{attribute 'linkalways'} 
{attribute 'no_explicit_call' := 'This FB is a CLASS and must be accessed using methods or properties'}
{attribute 'enable_dynamic_creation'}
FUNCTION_BLOCK FINAL ABS_ULINT EXTENDS Node
VAR
	in : _ULINT(0);
	out : _ULINT(0);
END_VAR

METHOD PUBLIC Clone : I_Node
VAR
	pNode : POINTER TO ABS_ULINT;
END_VAR
pNode := __NEW(ABS_ULINT);
Clone := pNode^;
END_METHOD

METHOD FB_init : BOOL
VAR_INPUT
	bInitRetains : BOOL; // if TRUE, the retain variables are initialized (warm start / cold start)
	bInCopyCode : BOOL;  // if TRUE, the instance afterwards gets moved into the copy code (online change)
END_VAR
AddInput('in',THIS^.in);
AddOutput('out', THIS^.out);
END_METHOD

METHOD PROTECTED OnExecute
VAR
END_VAR
out.Value := ABS(in.Value);
END_METHOD

END_FUNCTION_BLOCK

(* stored: Version 1.1.0.1, ProductVersion 3.1.4024.15
   POU ABS_ULINT: Id {d9e94608-85d9-4704-aef5-600e84c92692}, SpecialFunc None
   Folder Constructor: Id {b89a9a35-a5c0-4751-a23a-8c3e69466e39}
   Method Clone: Id {8666aac5-0a1a-49e8-aae3-2f59925bd958}
   Method FB_init: Id {30dfa24d-4c2c-43c3-8ef5-30a28923280d}
   Method OnExecute: Id {91a44e4e-c82d-4cf5-9a9b-6013f8673645} *)
